{attribute addProperty BoxType "KL1904"}
{attribute addProperty Id "Channel_1Channel_D8611DE600"}
{attribute addProperty CRC "1578653816"}
{attribute addProperty SizeInBites "0"}
{attribute addProperty SizeInBytes "0"}
TYPE KL1904_5E185878 :
STRUCT
	{attribute addProperty Name "Channel_1"}
	Channel_1 : Channel_D8611DE6;
END_STRUCT
END_TYPE

(* stored: Version 1.2.0.0, ProductVersion 3.1.4024.9
   DUT KL1904_5E185878: Id {b0e30e54-c9eb-484f-bb0d-ece9ca914279} *)
